PROGRAM PRG_TEST
VAR
	Motion	: MotionTest;
	NC		: NcParameterTest;
	XML		: XmlHandler_Test;
END_VAR

Motion();
NC();
XML();

END_PROGRAM

(* stored: Version 1.1.0.1
   POU PRG_TEST: Id {074b34d7-23f1-46e6-ab5c-dcdee3c6384a}, SpecialFunc None *)
